{attribute 'GeneratedUsingTerminal: EL7342-0000-0016'}
{attribute addProperty BoxType "EL7342-0000-0016"}
{attribute addProperty Id "Latch_extern_validBOOL1Set_counter_doneBOOL1Counter_underflowBOOL1Counter_overflowBOOL1Extrapolation_stallBOOL1Status_of_input_ABOOL1Status_of_input_BBOOL1Status_of_extern_latchBOOL1Sync_errorBOOL1TxPDO_ToggleBOOL1"}
{attribute addProperty CRC "808828462"}
{attribute addProperty Size "10"}
TYPE Status_3035BE2E :
STRUCT
	{attribute addProperty Name "Latch_extern_valid"}
	Latch_extern_valid : BOOL;
	{attribute addProperty Name "Set_counter_done"}
	Set_counter_done : BOOL;
	{attribute addProperty Name "Counter_underflow"}
	Counter_underflow : BOOL;
	{attribute addProperty Name "Counter_overflow"}
	Counter_overflow : BOOL;
	{attribute addProperty Name "Extrapolation_stall"}
	Extrapolation_stall : BOOL;
	{attribute addProperty Name "Status_of_input_A"}
	Status_of_input_A : BOOL;
	{attribute addProperty Name "Status_of_input_B"}
	Status_of_input_B : BOOL;
	{attribute addProperty Name "Status_of_extern_latch"}
	Status_of_extern_latch : BOOL;
	{attribute addProperty Name "Sync_error"}
	Sync_error : BOOL;
	{attribute addProperty Name "TxPDO_Toggle"}
	TxPDO_Toggle : BOOL;
END_STRUCT
END_TYPE

(* stored: Version 1.2.0.0, ProductVersion 3.1.4024.9
   DUT Status_3035BE2E: Id {bbb66758-8e5b-45ea-858f-658c4a701071} *)
